(* Logix 5000 project; controller HP_SSC01 vendor 1 type 14 code 67 rev 17.7; software revision 17.01; part 2 of 15 *)
(* tags used below, declared in another part *)
   A_C1_0300 : ALIAS FOR C1_FaultStandard.0;
   A_C1_0301 : ALIAS FOR C1_FaultStandard.1;
   A_C1_0302 : ALIAS FOR C1_FaultStandard.2;
   A_C1_0303 : ALIAS FOR C1_FaultStandard.3;
   A_C1_0305 : ALIAS FOR C1_FaultStandard.5;
   A_C1_0309 : ALIAS FOR C1_FaultStandard.9;
   A_C1_0310 : ALIAS FOR C1_FaultStandard.10;
   A_C1_0311 : ALIAS FOR C1_FaultStandard.11;
   A_C1_0312 : ALIAS FOR C1_FaultStandard.12;
   A_C1_0313 : ALIAS FOR C1_FaultStandard.13;
   A_C1_0314 : ALIAS FOR C1_FaultStandard.14;
   A_C1_0315 : ALIAS FOR C1_FaultStandard.15;
   A_C1_0317 : ALIAS FOR C1_FaultStandard.17;
   A_C1_0319 : ALIAS FOR C1_FaultStandard.19;
   A_C1_0321 : ALIAS FOR C1_FaultStandard.21;
   A_C1_0322 : ALIAS FOR C1_FaultStandard.22;
   A_C1_0323 : ALIAS FOR C1_FaultStandard.23;
   A_C1_0324 : ALIAS FOR C1_FaultStandard.24;
   A_C1_0325 : ALIAS FOR C1_FaultStandard.25;
   A_C1_0327 : ALIAS FOR C1_FaultStandard.27;
   A_C1_0328 : ALIAS FOR C1_FaultStandard.28;
   A_C1_0329 : ALIAS FOR C1_FaultStandard.29;
   A_C1_0330 : ALIAS FOR C1_FaultStandard.30;
   A_C1_0331 : ALIAS FOR C1_FaultStandard.31;
   A_C1_0404 : ALIAS FOR C1_Warning.4;
   A_C1_0406 : ALIAS FOR C1_Warning.6;
   A_C1_0407 : ALIAS FOR C1_Warning.7;
   A_C1_0408 : ALIAS FOR C1_Warning.8;
   A_C1_0409 : ALIAS FOR C1_Warning.9;
   A_C1_0412 : ALIAS FOR C1_Warning.12;
   A_C1_0413 : ALIAS FOR C1_Warning.13;
   A_C1_0414 : ALIAS FOR C1_Warning.14;
   A_C1_0415 : ALIAS FOR C1_Warning.15;
   A_C1_0416 : ALIAS FOR C1_Warning.16;
   A_C1_0424 : ALIAS FOR C1_Warning.24;
   A_C1_0427 : ALIAS FOR C1_Warning.27;
   A_C1_0428 : ALIAS FOR C1_Warning.28;
   A_C1_0430 : ALIAS FOR C1_Warning.30;
   C1 : AXIS_SERVO_DRIVE;
   C1_32HourTimers : TIMER[8];
   C1_All_DLY_OK : BOOL;
   C1_BrakeSequenceInProcess : BOOL;
   C1_BrakeTest : BOOL;
   C1_BrakeTestEndPosition : REAL;
   C1_BrakeTestFailed : BOOL;
   C1_BrakeTestLocalDisable : BOOL;
   C1_BrakeTestMAJ01 : MOTION_INSTRUCTION;
   C1_BrakeTestMessageNumber : DINT;
   C1_BrakeTestONS : BOOL;
   C1_BrakeTestSelected : BOOL;
   C1_BrakeTestSequence : DINT;
   C1_BrakeTestSequenceAlarms : DINT;
   C1_BrakeTestSequenceAlarmTimer : TIMER[16];
   C1_BrakeTestSequenceONS : DINT;
   C1_BrakeTestStartPosition : REAL;
   C1_BrakeTestStoppingDistance : REAL;
   C1_BrakeTestTimerHoldVel : TIMER;
   C1_BrakeTestWarning : BOOL;
   C1_DisableTimer : TIMER;
   C1_DumpTest : BOOL;
   C1_DumpValveFailedOff : BOOL;
   C1_DumpValveFailedOn : BOOL;
   C1_DumpValveMessageNumber : DINT;
   C1_DumpValveTestDelay : TIMER[4];
   C1_DumpValveTestDelay2 : TIMER;
   C1_DumpValveTestSelected : BOOL;
   C1_DumpValveTestSequence : DINT;
   C1_DumpValveTestSequenceAlarms : DINT;
   C1_DumpValveTestSequenceAlarmTimer : TIMER[16];
   C1_EncoderCounts : DINT;
   C1_EncoderCountsRaw : ALIAS FOR C1_RIO_AENT:3:I.PresentData;
   C1_EncoderDegree : REAL;
   C1_FaultDebounce : TIMER[16];
   C1_FaultHoldTimer : TIMER[8];
   C1_FaultHomeSwitchNotFound : BOOL;
   C1_FaultStandard : DINT;
   C1_HomeInputStatus : BOOL;
   C1_HomeSequence : DINT;
   C1_HomeSequenceAlarms : DINT;
   C1_HomeSwitchFaultK7KFailedOff : BOOL;
   C1_HomeSwitchFaultK7KFailedOn : BOOL;
   C1_HomeSwitchFaultSafeFailedOff : BOOL;
   C1_HomeSwitchFaultSafeFailedOn : BOOL;
   C1_IndexEnable : BOOL;
   C1_JogEnable : BOOL;
   C1_LIM_ALARM_B : ALIAS FOR C1_RIO_AENT:I.Data[1].0;
   C1_MaintEnable : BOOL;
   C1_MotorActualPositionX1000 : DINT;
   C1_MotorAverageVelocityX1000 : DINT;
   C1_MotorFan : ALIAS FOR C1_RIO_AENT:O.Data[2].0;
   C1_MSF : MOTION_INSTRUCTION;
   C1_MSO : MOTION_INSTRUCTION;
   C1_OIT_Current : DINT;
   C1_ONS_Fault : DINT;
   C1_RemoteBrakeAndHomeSequenceAlarms : DINT;
   C1_RemoteBrakeTestCMD : BOOL;
   C1_RemoteDumpTestCMD : BOOL;
   C1_ServoActionStatusOffDelay : TIMER;
   C1_ServoActionStatusOnDelay : TIMER;
   C1_ServoFanOverload : ALIAS FOR C1_RIO_AENT:I.Data[1].2;
   C1_SS_LocalRemote_1_IsRemote : ALIAS FOR C1_RIO_AENT:1:I.3;
   C1_SS_RemoteMode : BOOL;
   C1_Warning : DINT;
   C1DumpValveTestSequenceONS : DINT;
   RCS_CMD_RunInAuto : BOOL;
   RCS_SyncMotionEnable : BOOL;
   S_C1_EncoderPositionDegree : DINT;
   S_C1_ExecutePB : BOOL;
   S_C1_FaultReset : BOOL;
   S_C1_ModeLocal : BOOL;
   S_C1_ModeRemote : BOOL;
   S_C1_MotionEnabled : BOOL;
   S_C1_MSTOP_InputOK : BOOL;
   S_C1_NearOnPath : BOOL;
   S_C1_OffPath : BOOL;
   S_C1_OIT_FaultReset : BOOL;
   S_C1_OutputEnable : BOOL;
   S_C1_PressureOK : ALIAS FOR C1_Safe:I.Pt05Data;
   S_C1_SAFETY_ENABLE_1 : ALIAS FOR C1_Safe:O.Pt00Data;
   S_C1_SAFETY_ENABLE_2 : ALIAS FOR C1_Safe:O.Pt01Data;
   S_C1_Stop1_OK : BOOL;
   S_RCS_CMD_FaultReset : BOOL;
   STS_Enable_Rail : DINT;
   ZZZ_DIAG_A_C1_0302 : BOOL;
   ZZZ_DIAG_C1_AxisFault : DINT;
   ZZZ_DIAG_C1_AxisStatus : DINT;
   ZZZ_DIAG_C1_EnableRail : DINT;
   ZZZ_DIAG_C1_MotionStatus : DINT;
   ZZZ_DIAG_C1_MSF : MOTION_INSTRUCTION;
   ZZZ_DIAG_C1_MSO : MOTION_INSTRUCTION;
   ZZZ_DIAG_C1_OneTimeOnly : BOOL;
   ZZZ_DIAG_C1_OutputEnable : BOOL;
   ZZZ_DIAG_C1_OutputEnable_ACC : DINT;
   ZZZ_DIAG_ONS : DINT;
   ZZZ_DIAG_S_C1_OutputEnableTON : TIMER;
   ZZZ_DIAG_S_C1_SAFETY_ENABLE_1 : BOOL;
   ZZZ_DIAG_S_C1_SAFETY_ENABLE_2 : BOOL;

PROGRAM Carousel1   (* main routine C100_Main *)
VAR
   SCRV_01 : S_CURVE := (In := 26.237068, AccelRate := 100000.0, DecelRate := 100000.0, JerkRate := 100.0, RTSTime := 1, S_Mode := 1, Out := 25.846554, Rate := 8.784333, DeltaT := 0.01);
   zzz_Test10 : BOOL;
   zzz_Test11 : BOOL;
   zzz_TestOffset : DINT := 1000;
   zzz_TestWord10 : DINT;
END_VAR

ROUTINE C100_Main   (* ladder *)
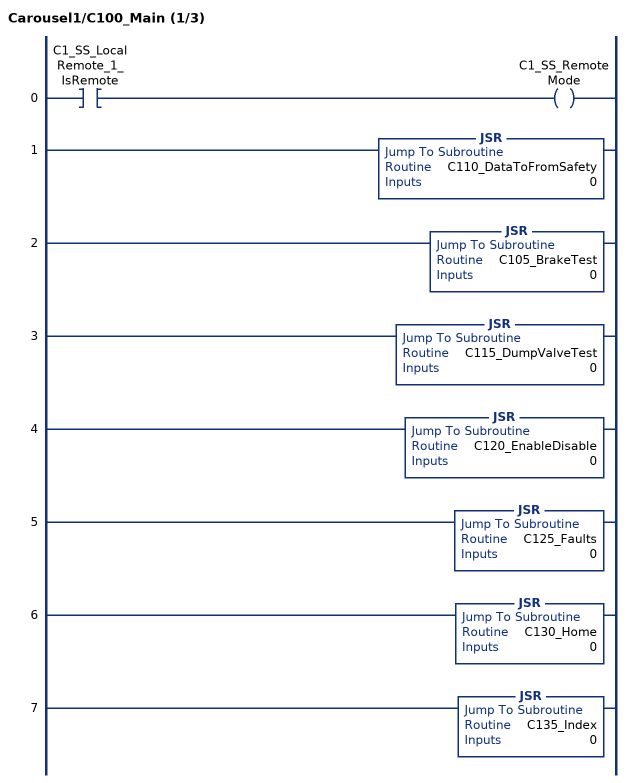
   0: XIC(C1_SS_LocalRemote_1_IsRemote)OTE(C1_SS_RemoteMode);
   1: JSR(C110_DataToFromSafety,0);
   2: JSR(C105_BrakeTest,0);
   3: JSR(C115_DumpValveTest,0);
   4: JSR(C120_EnableDisable,0);
   5: JSR(C125_Faults,0);
   6: JSR(C130_Home,0);
   7: JSR(C135_Index,0);
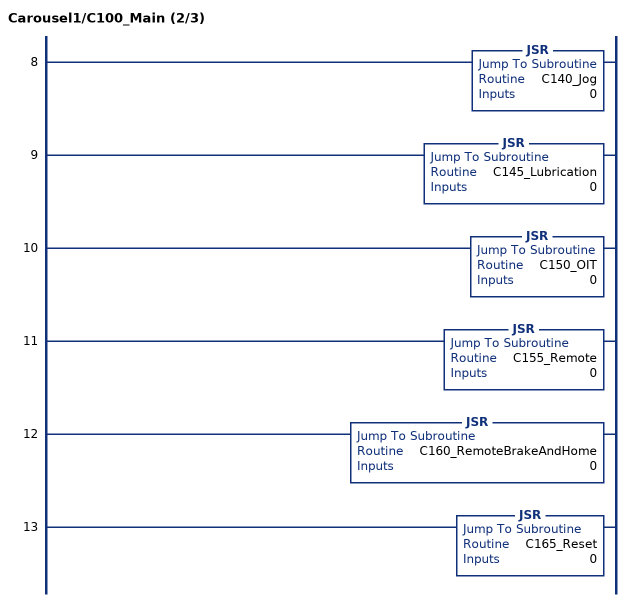
   8: JSR(C140_Jog,0);
   9: JSR(C145_Lubrication,0);
   10: JSR(C150_OIT,0);
   11: JSR(C155_Remote,0);
   12: JSR(C160_RemoteBrakeAndHome,0);
   13: JSR(C165_Reset,0);
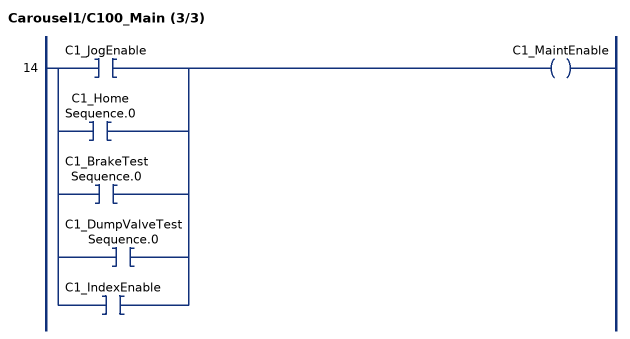
   14: [XIC(C1_JogEnable) ,XIC(C1_HomeSequence.0) ,XIC(C1_BrakeTestSequence.0) ,XIC(C1_DumpValveTestSequence.0) ,XIC(C1_IndexEnable) ]OTE(C1_MaintEnable);
END_ROUTINE

ROUTINE C105_BrakeTest   (* ladder *)
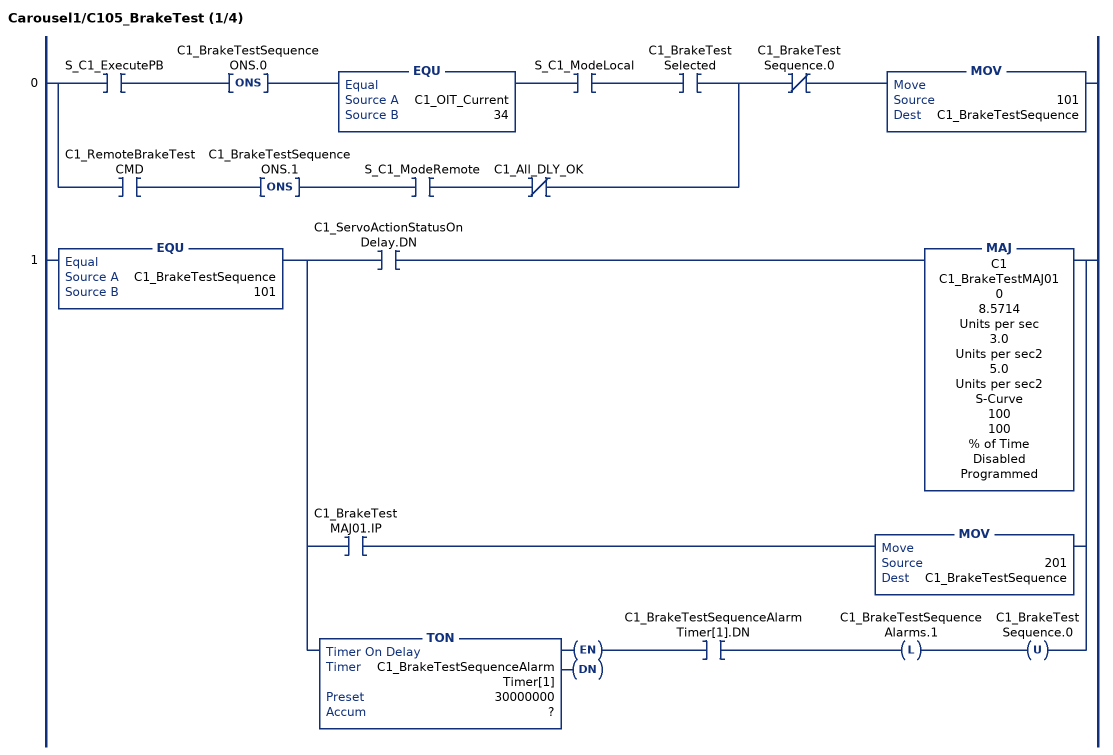
   0: [XIC(S_C1_ExecutePB) ONS(C1_BrakeTestSequenceONS.0) EQU(C1_OIT_Current,34) XIC(S_C1_ModeLocal) XIC(C1_BrakeTestSelected) ,XIC(C1_RemoteBrakeTestCMD) ONS(C1_BrakeTestSequenceONS.1) XIC(S_C1_ModeRemote) XIO(C1_All_DLY_OK) ]XIO(C1_BrakeTestSequence.0)MOV(101,C1_BrakeTestSequence);
   1: EQU(C1_BrakeTestSequence,101)[XIC(C1_ServoActionStatusOnDelay.DN) MAJ(C1,C1_BrakeTestMAJ01,0,8.5714,Units per sec,3.0,Units per sec2,5.0,Units per sec2,S-Curve,100,100,% of Time,Disabled,Programmed) ,XIC(C1_BrakeTestMAJ01.IP) MOV(201,C1_BrakeTestSequence) ,TON(C1_BrakeTestSequenceAlarmTimer[1],?,?) XIC(C1_BrakeTestSequenceAlarmTimer[1].DN) OTL(C1_BrakeTestSequenceAlarms.1) OTU(C1_BrakeTestSequence.0) ];
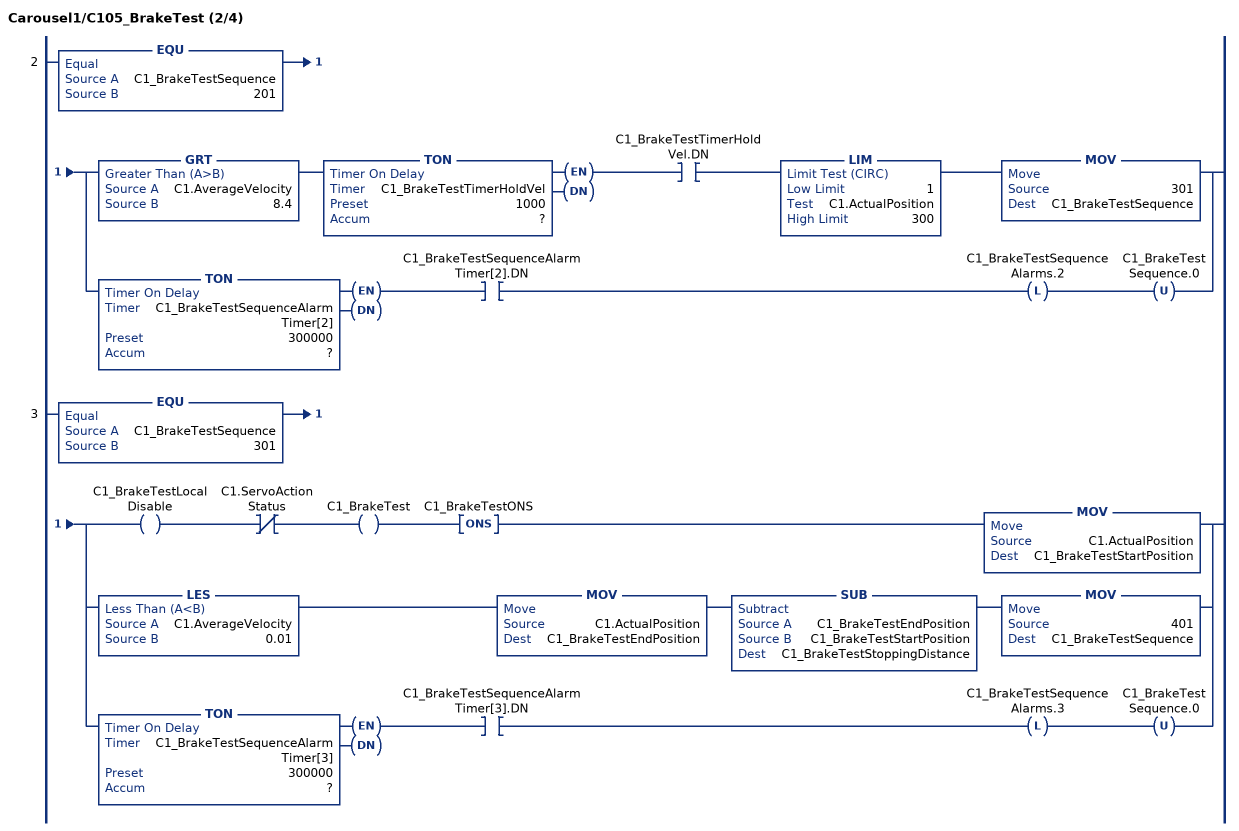
   2: EQU(C1_BrakeTestSequence,201)[GRT(C1.AverageVelocity,8.4) TON(C1_BrakeTestTimerHoldVel,?,?) XIC(C1_BrakeTestTimerHoldVel.DN) LIM(1,C1.ActualPosition,300) MOV(301,C1_BrakeTestSequence) ,TON(C1_BrakeTestSequenceAlarmTimer[2],?,?) XIC(C1_BrakeTestSequenceAlarmTimer[2].DN) OTL(C1_BrakeTestSequenceAlarms.2) OTU(C1_BrakeTestSequence.0) ];
   3: EQU(C1_BrakeTestSequence,301)[OTE(C1_BrakeTestLocalDisable) XIO(C1.ServoActionStatus) OTE(C1_BrakeTest) ONS(C1_BrakeTestONS) MOV(C1.ActualPosition,C1_BrakeTestStartPosition) ,LES(C1.AverageVelocity,0.01) MOV(C1.ActualPosition,C1_BrakeTestEndPosition) SUB(C1_BrakeTestEndPosition,C1_BrakeTestStartPosition,C1_BrakeTestStoppingDistance) MOV(401,C1_BrakeTestSequence) ,TON(C1_BrakeTestSequenceAlarmTimer[3],?,?) XIC(C1_BrakeTestSequenceAlarmTimer[3].DN) OTL(C1_BrakeTestSequenceAlarms.3) OTU(C1_BrakeTestSequence.0) ];
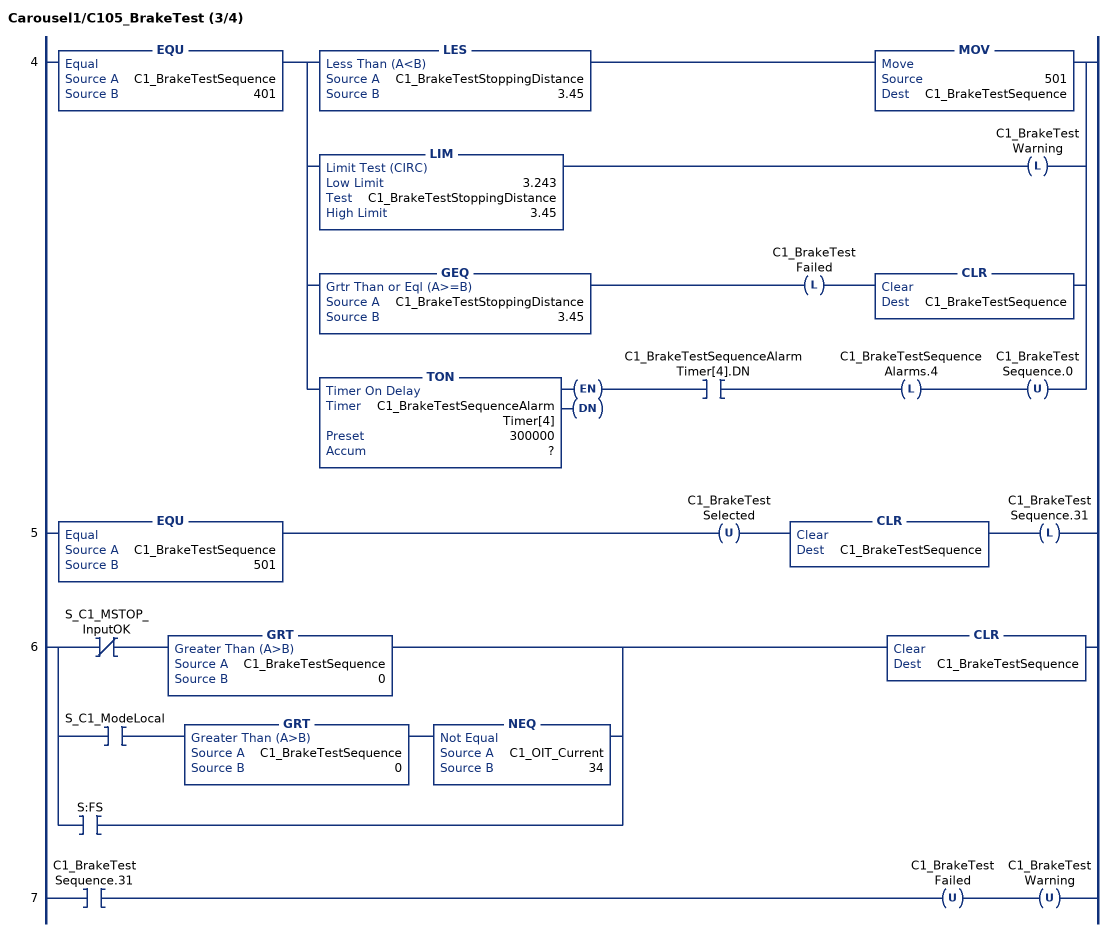
   4: EQU(C1_BrakeTestSequence,401)[LES(C1_BrakeTestStoppingDistance,3.45) MOV(501,C1_BrakeTestSequence) ,LIM(3.243,C1_BrakeTestStoppingDistance,3.45) OTL(C1_BrakeTestWarning) ,GEQ(C1_BrakeTestStoppingDistance,3.45) OTL(C1_BrakeTestFailed) CLR(C1_BrakeTestSequence) ,TON(C1_BrakeTestSequenceAlarmTimer[4],?,?) XIC(C1_BrakeTestSequenceAlarmTimer[4].DN) OTL(C1_BrakeTestSequenceAlarms.4) OTU(C1_BrakeTestSequence.0) ];
   5: EQU(C1_BrakeTestSequence,501)OTU(C1_BrakeTestSelected)CLR(C1_BrakeTestSequence)OTL(C1_BrakeTestSequence.31);
   6: [XIO(S_C1_MSTOP_InputOK) GRT(C1_BrakeTestSequence,0) ,XIC(S_C1_ModeLocal) GRT(C1_BrakeTestSequence,0) NEQ(C1_OIT_Current,34) ,XIC(S:FS) ]CLR(C1_BrakeTestSequence);
   7: XIC(C1_BrakeTestSequence.31)OTU(C1_BrakeTestFailed)OTU(C1_BrakeTestWarning);
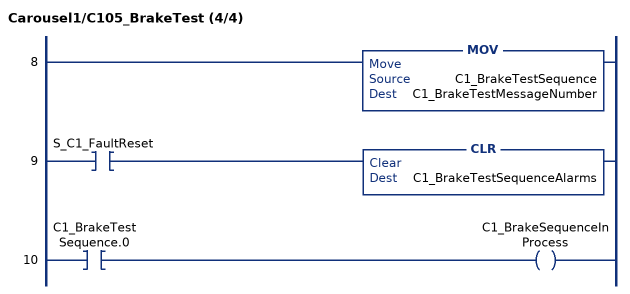
   8: MOV(C1_BrakeTestSequence,C1_BrakeTestMessageNumber);
   9: XIC(S_C1_FaultReset)CLR(C1_BrakeTestSequenceAlarms);
   10: XIC(C1_BrakeTestSequence.0)OTE(C1_BrakeSequenceInProcess);
END_ROUTINE

ROUTINE C110_DataToFromSafety   (* ladder *)
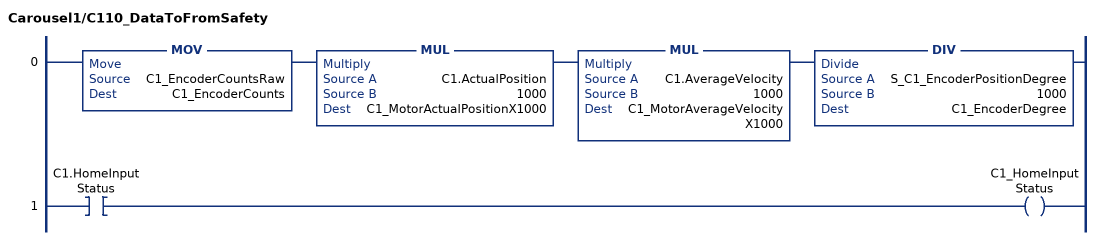
   0: MOV(C1_EncoderCountsRaw,C1_EncoderCounts)MUL(C1.ActualPosition,1000,C1_MotorActualPositionX1000)MUL(C1.AverageVelocity,1000,C1_MotorAverageVelocityX1000)DIV(S_C1_EncoderPositionDegree,1000,C1_EncoderDegree);
   1: XIC(C1.HomeInputStatus)OTE(C1_HomeInputStatus);
END_ROUTINE

ROUTINE C115_DumpValveTest   (* ladder *)
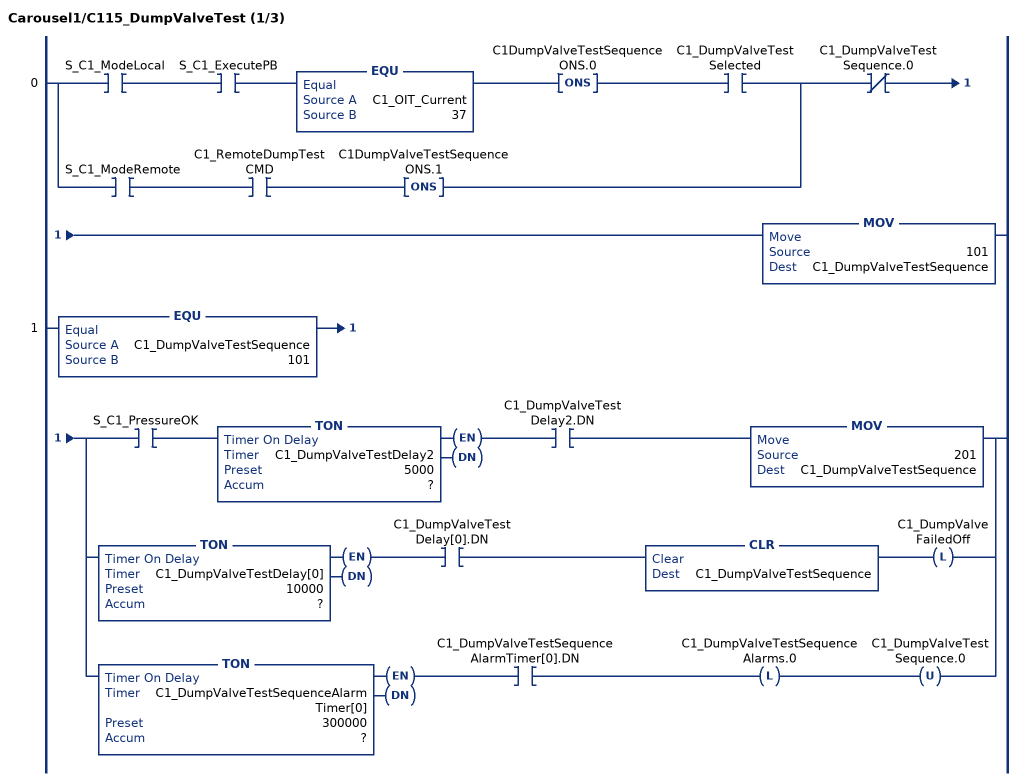
   0: [XIC(S_C1_ModeLocal) XIC(S_C1_ExecutePB) EQU(C1_OIT_Current,37) ONS(C1DumpValveTestSequenceONS.0) XIC(C1_DumpValveTestSelected) ,XIC(S_C1_ModeRemote) XIC(C1_RemoteDumpTestCMD) ONS(C1DumpValveTestSequenceONS.1) ]XIO(C1_DumpValveTestSequence.0)MOV(101,C1_DumpValveTestSequence);
   1: EQU(C1_DumpValveTestSequence,101)[XIC(S_C1_PressureOK) TON(C1_DumpValveTestDelay2,?,?) XIC(C1_DumpValveTestDelay2.DN) MOV(201,C1_DumpValveTestSequence) ,TON(C1_DumpValveTestDelay[0],?,?) XIC(C1_DumpValveTestDelay[0].DN) CLR(C1_DumpValveTestSequence) OTL(C1_DumpValveFailedOff) ,TON(C1_DumpValveTestSequenceAlarmTimer[0],?,?) XIC(C1_DumpValveTestSequenceAlarmTimer[0].DN) OTL(C1_DumpValveTestSequenceAlarms.0) OTU(C1_DumpValveTestSequence.0) ];
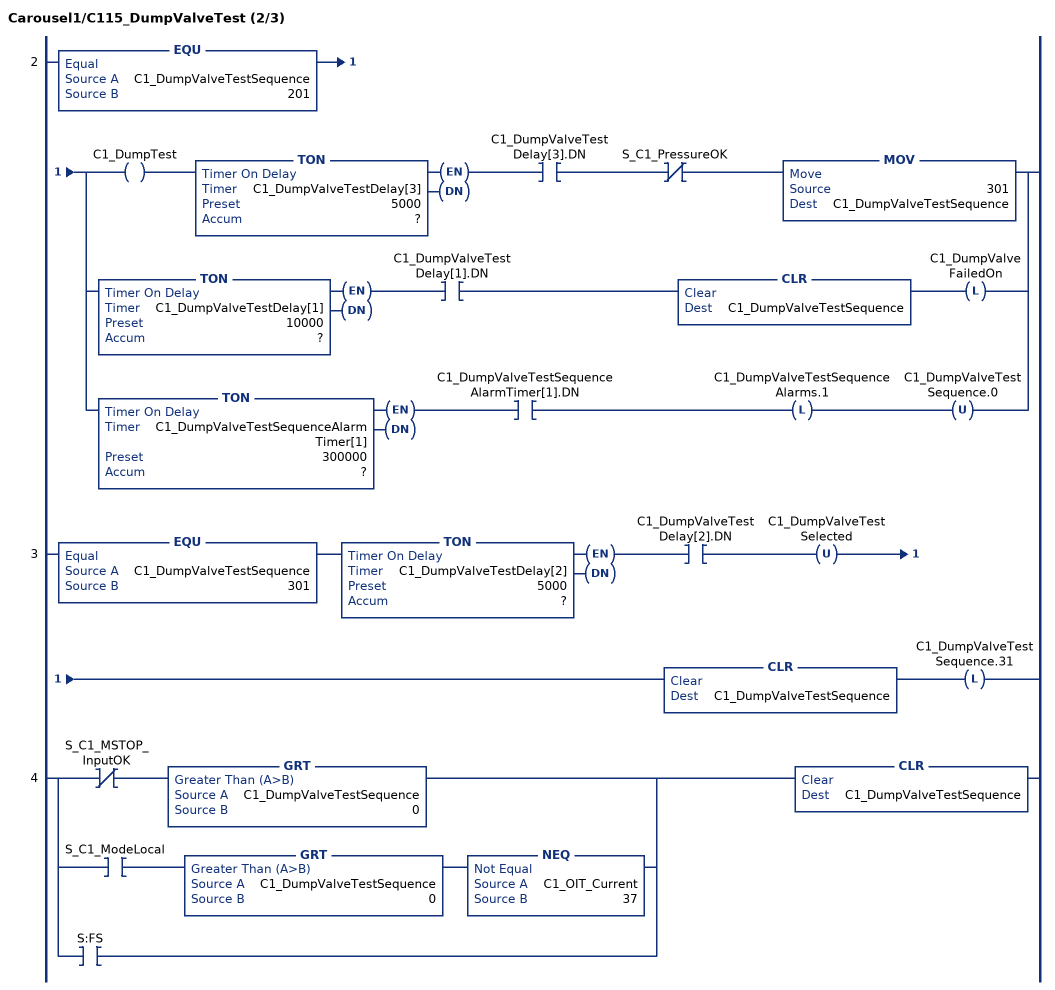
   2: EQU(C1_DumpValveTestSequence,201)[OTE(C1_DumpTest) TON(C1_DumpValveTestDelay[3],?,?) XIC(C1_DumpValveTestDelay[3].DN) XIO(S_C1_PressureOK) MOV(301,C1_DumpValveTestSequence) ,TON(C1_DumpValveTestDelay[1],?,?) XIC(C1_DumpValveTestDelay[1].DN) CLR(C1_DumpValveTestSequence) OTL(C1_DumpValveFailedOn) ,TON(C1_DumpValveTestSequenceAlarmTimer[1],?,?) XIC(C1_DumpValveTestSequenceAlarmTimer[1].DN) OTL(C1_DumpValveTestSequenceAlarms.1) OTU(C1_DumpValveTestSequence.0) ];
   3: EQU(C1_DumpValveTestSequence,301)TON(C1_DumpValveTestDelay[2],?,?)XIC(C1_DumpValveTestDelay[2].DN)OTU(C1_DumpValveTestSelected)CLR(C1_DumpValveTestSequence)OTL(C1_DumpValveTestSequence.31);
   4: [XIO(S_C1_MSTOP_InputOK) GRT(C1_DumpValveTestSequence,0) ,XIC(S_C1_ModeLocal) GRT(C1_DumpValveTestSequence,0) NEQ(C1_OIT_Current,37) ,XIC(S:FS) ]CLR(C1_DumpValveTestSequence);
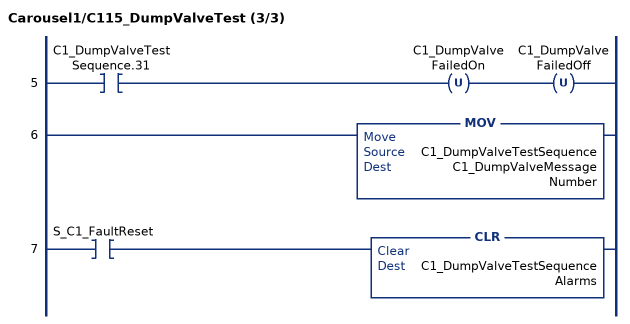
   5: XIC(C1_DumpValveTestSequence.31)OTU(C1_DumpValveFailedOn)OTU(C1_DumpValveFailedOff);
   6: MOV(C1_DumpValveTestSequence,C1_DumpValveMessageNumber);
   7: XIC(S_C1_FaultReset)CLR(C1_DumpValveTestSequenceAlarms);
END_ROUTINE

ROUTINE C120_EnableDisable   (* ladder *)
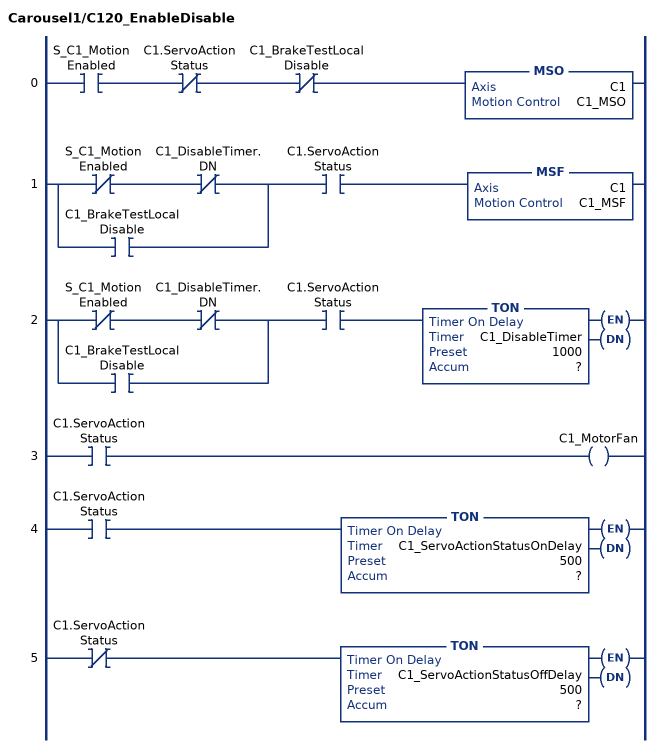
   0: XIC(S_C1_MotionEnabled)XIO(C1.ServoActionStatus)XIO(C1_BrakeTestLocalDisable)MSO(C1,C1_MSO);
   1: [XIO(S_C1_MotionEnabled) XIO(C1_DisableTimer.DN) ,XIC(C1_BrakeTestLocalDisable) ]XIC(C1.ServoActionStatus)MSF(C1,C1_MSF);
   2: [XIO(S_C1_MotionEnabled) XIO(C1_DisableTimer.DN) ,XIC(C1_BrakeTestLocalDisable) ]XIC(C1.ServoActionStatus)TON(C1_DisableTimer,?,?);
   3: XIC(C1.ServoActionStatus)OTE(C1_MotorFan);
   4: XIC(C1.ServoActionStatus)TON(C1_ServoActionStatusOnDelay,?,?);
   5: XIO(C1.ServoActionStatus)TON(C1_ServoActionStatusOffDelay,?,?);
END_ROUTINE

ROUTINE C125_Faults   (* ladder *)
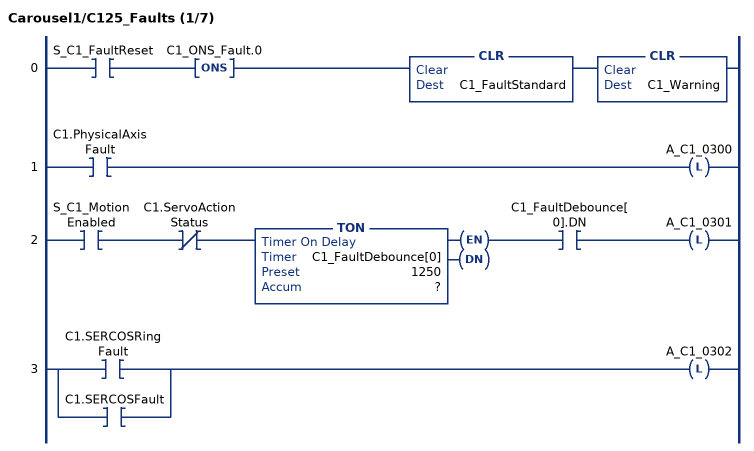
   0: XIC(S_C1_FaultReset)ONS(C1_ONS_Fault.0)CLR(C1_FaultStandard)CLR(C1_Warning);
   1: XIC(C1.PhysicalAxisFault)OTL(A_C1_0300);
   2: XIC(S_C1_MotionEnabled)XIO(C1.ServoActionStatus)TON(C1_FaultDebounce[0],?,?)XIC(C1_FaultDebounce[0].DN)OTL(A_C1_0301);
   3: [XIC(C1.SERCOSRingFault) ,XIC(C1.SERCOSFault) ]OTL(A_C1_0302);
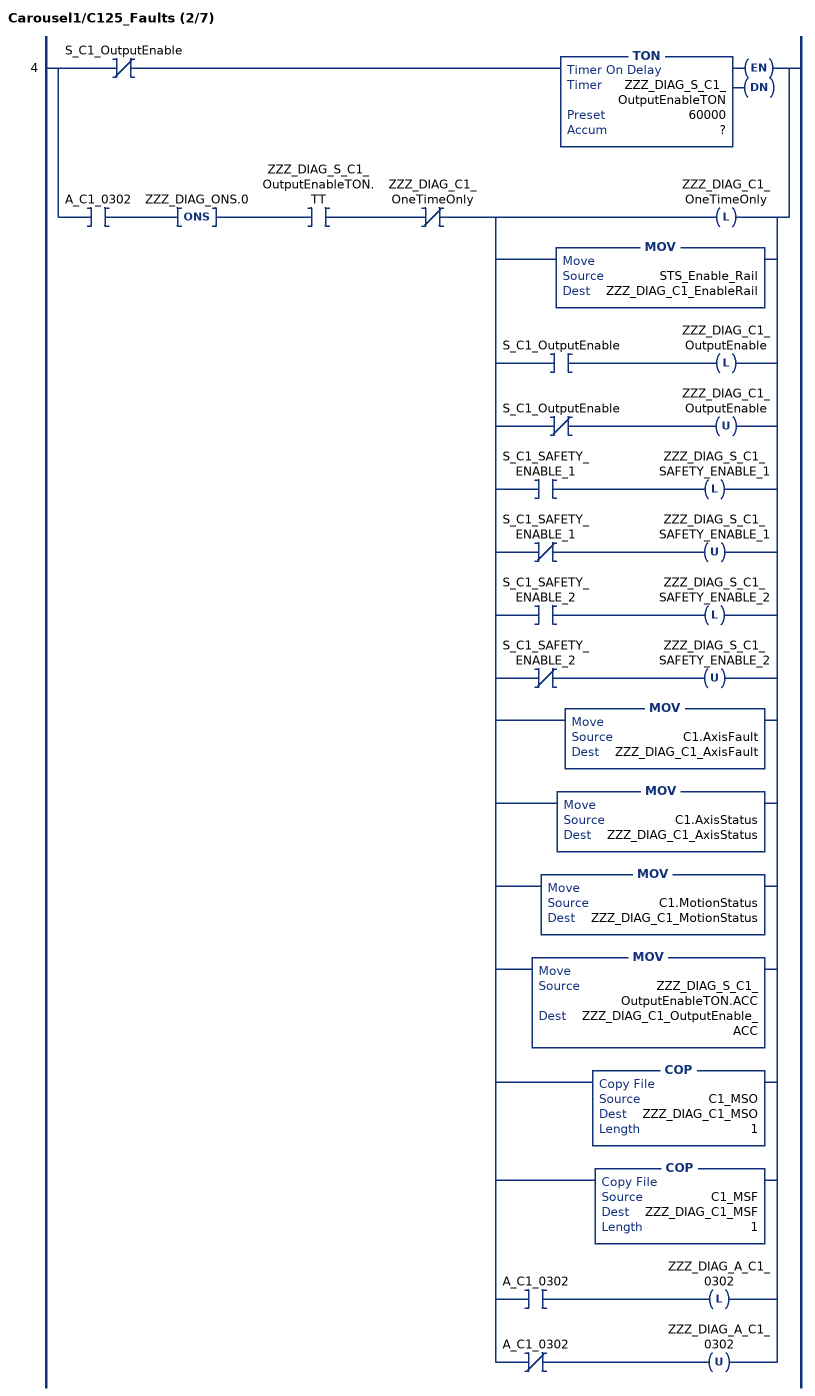
   4: [XIO(S_C1_OutputEnable) TON(ZZZ_DIAG_S_C1_OutputEnableTON,?,?) ,XIC(A_C1_0302) ONS(ZZZ_DIAG_ONS.0) XIC(ZZZ_DIAG_S_C1_OutputEnableTON.TT) XIO(ZZZ_DIAG_C1_OneTimeOnly) [OTL(ZZZ_DIAG_C1_OneTimeOnly) ,MOV(STS_Enable_Rail,ZZZ_DIAG_C1_EnableRail) ,XIC(S_C1_OutputEnable) OTL(ZZZ_DIAG_C1_OutputEnable) ,XIO(S_C1_OutputEnable) OTU(ZZZ_DIAG_C1_OutputEnable) ,XIC(S_C1_SAFETY_ENABLE_1) OTL(ZZZ_DIAG_S_C1_SAFETY_ENABLE_1) ,XIO(S_C1_SAFETY_ENABLE_1) OTU(ZZZ_DIAG_S_C1_SAFETY_ENABLE_1) ,XIC(S_C1_SAFETY_ENABLE_2) OTL(ZZZ_DIAG_S_C1_SAFETY_ENABLE_2) ,XIO(S_C1_SAFETY_ENABLE_2) OTU(ZZZ_DIAG_S_C1_SAFETY_ENABLE_2) ,MOV(C1.AxisFault,ZZZ_DIAG_C1_AxisFault) ,MOV(C1.AxisStatus,ZZZ_DIAG_C1_AxisStatus) ,MOV(C1.MotionStatus,ZZZ_DIAG_C1_MotionStatus) ,MOV(ZZZ_DIAG_S_C1_OutputEnableTON.ACC,ZZZ_DIAG_C1_OutputEnable_ACC) ,COP(C1_MSO,ZZZ_DIAG_C1_MSO,1) ,COP(C1_MSF,ZZZ_DIAG_C1_MSF,1) ,XIC(A_C1_0302) OTL(ZZZ_DIAG_A_C1_0302) ,XIO(A_C1_0302) OTU(ZZZ_DIAG_A_C1_0302) ] ];
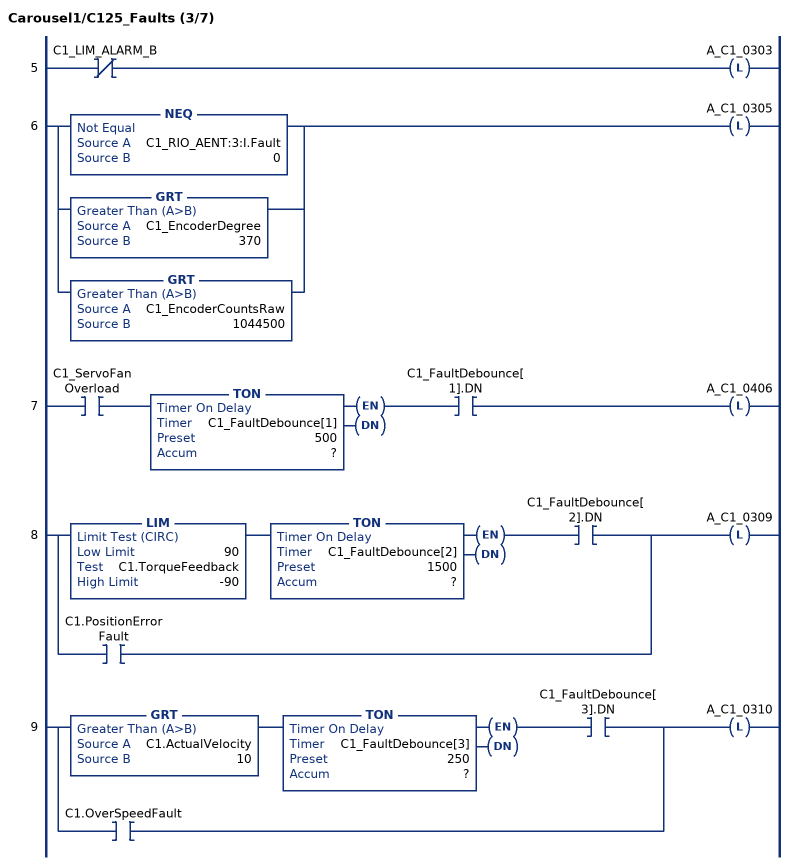
   5: XIO(C1_LIM_ALARM_B)OTL(A_C1_0303);
   6: [NEQ(C1_RIO_AENT:3:I.Fault,0) ,GRT(C1_EncoderDegree,370) ,GRT(C1_EncoderCountsRaw,1044500) ]OTL(A_C1_0305);
   7: XIC(C1_ServoFanOverload)TON(C1_FaultDebounce[1],?,?)XIC(C1_FaultDebounce[1].DN)OTL(A_C1_0406);
   8: [LIM(90,C1.TorqueFeedback,-90) TON(C1_FaultDebounce[2],?,?) XIC(C1_FaultDebounce[2].DN) ,XIC(C1.PositionErrorFault) ]OTL(A_C1_0309);
   9: [GRT(C1.ActualVelocity,10) TON(C1_FaultDebounce[3],?,?) XIC(C1_FaultDebounce[3].DN) ,XIC(C1.OverSpeedFault) ]OTL(A_C1_0310);
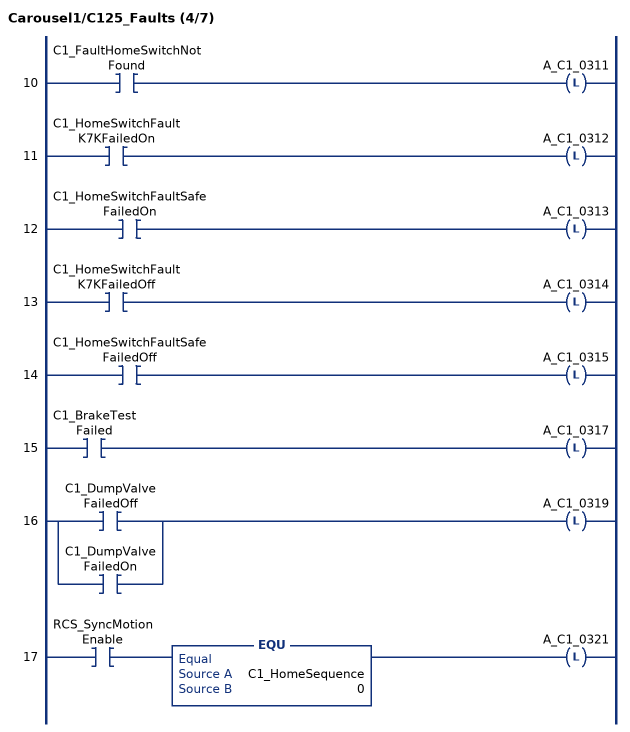
   10: XIC(C1_FaultHomeSwitchNotFound)OTL(A_C1_0311);
   11: XIC(C1_HomeSwitchFaultK7KFailedOn)OTL(A_C1_0312);
   12: XIC(C1_HomeSwitchFaultSafeFailedOn)OTL(A_C1_0313);
   13: XIC(C1_HomeSwitchFaultK7KFailedOff)OTL(A_C1_0314);
   14: XIC(C1_HomeSwitchFaultSafeFailedOff)OTL(A_C1_0315);
   15: XIC(C1_BrakeTestFailed)OTL(A_C1_0317);
   16: [XIC(C1_DumpValveFailedOff) ,XIC(C1_DumpValveFailedOn) ]OTL(A_C1_0319);
   17: XIC(RCS_SyncMotionEnable)EQU(C1_HomeSequence,0)OTL(A_C1_0321);
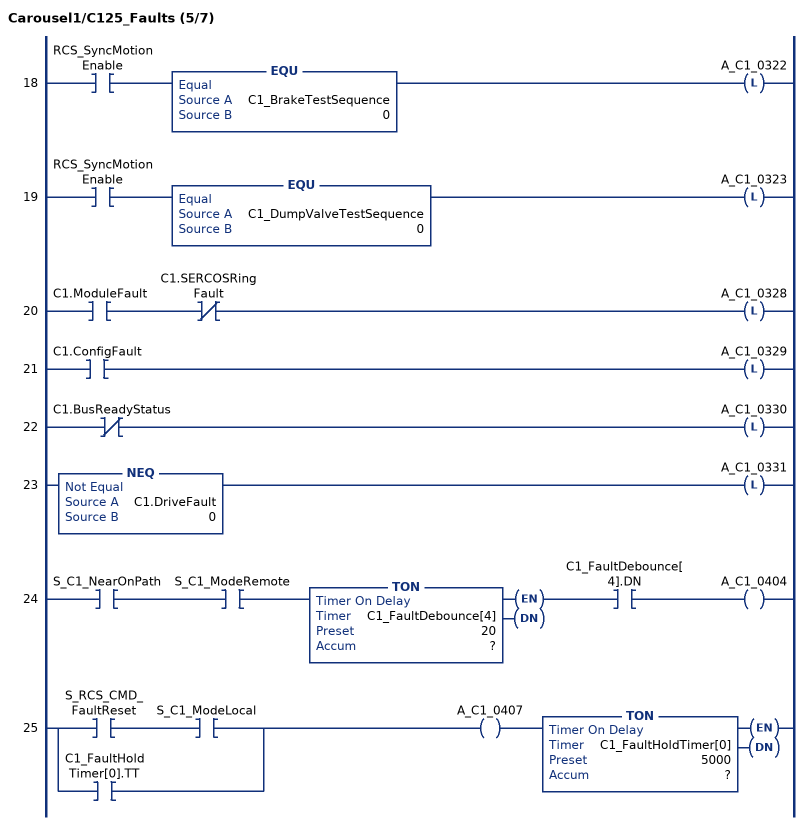
   18: XIC(RCS_SyncMotionEnable)EQU(C1_BrakeTestSequence,0)OTL(A_C1_0322);
   19: XIC(RCS_SyncMotionEnable)EQU(C1_DumpValveTestSequence,0)OTL(A_C1_0323);
   20: XIC(C1.ModuleFault)XIO(C1.SERCOSRingFault)OTL(A_C1_0328);
   21: XIC(C1.ConfigFault)OTL(A_C1_0329);
   22: XIO(C1.BusReadyStatus)OTL(A_C1_0330);
   23: NEQ(C1.DriveFault,0)OTL(A_C1_0331);
   24: XIC(S_C1_NearOnPath)XIC(S_C1_ModeRemote)TON(C1_FaultDebounce[4],?,?)XIC(C1_FaultDebounce[4].DN)OTE(A_C1_0404);
   25: [XIC(S_RCS_CMD_FaultReset) XIC(S_C1_ModeLocal) ,XIC(C1_FaultHoldTimer[0].TT) ]OTE(A_C1_0407)TON(C1_FaultHoldTimer[0],?,?);
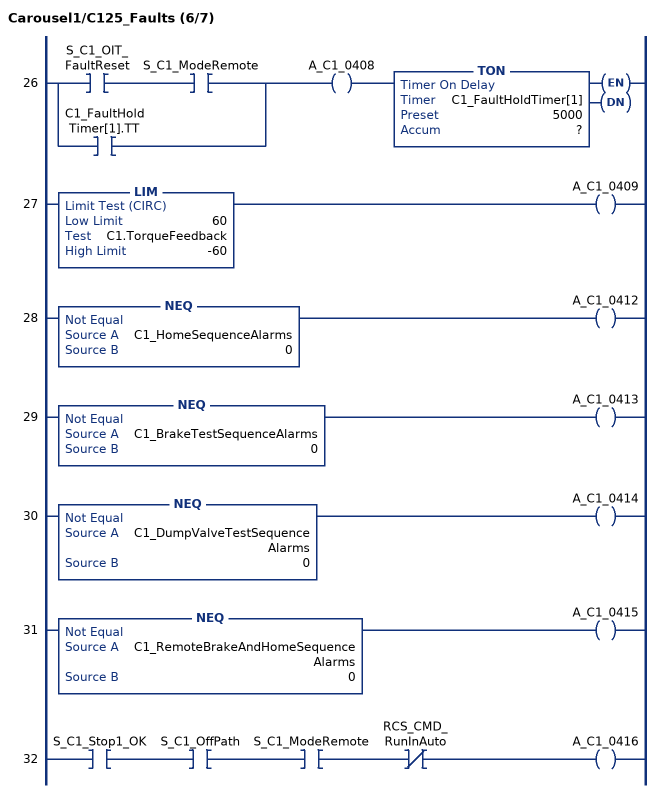
   26: [XIC(S_C1_OIT_FaultReset) XIC(S_C1_ModeRemote) ,XIC(C1_FaultHoldTimer[1].TT) ]OTE(A_C1_0408)TON(C1_FaultHoldTimer[1],?,?);
   27: LIM(60,C1.TorqueFeedback,-60)OTE(A_C1_0409);
   28: NEQ(C1_HomeSequenceAlarms,0)OTE(A_C1_0412);
   29: NEQ(C1_BrakeTestSequenceAlarms,0)OTE(A_C1_0413);
   30: NEQ(C1_DumpValveTestSequenceAlarms,0)OTE(A_C1_0414);
   31: NEQ(C1_RemoteBrakeAndHomeSequenceAlarms,0)OTE(A_C1_0415);
   32: XIC(S_C1_Stop1_OK)XIC(S_C1_OffPath)XIC(S_C1_ModeRemote)XIO(RCS_CMD_RunInAuto)OTE(A_C1_0416);
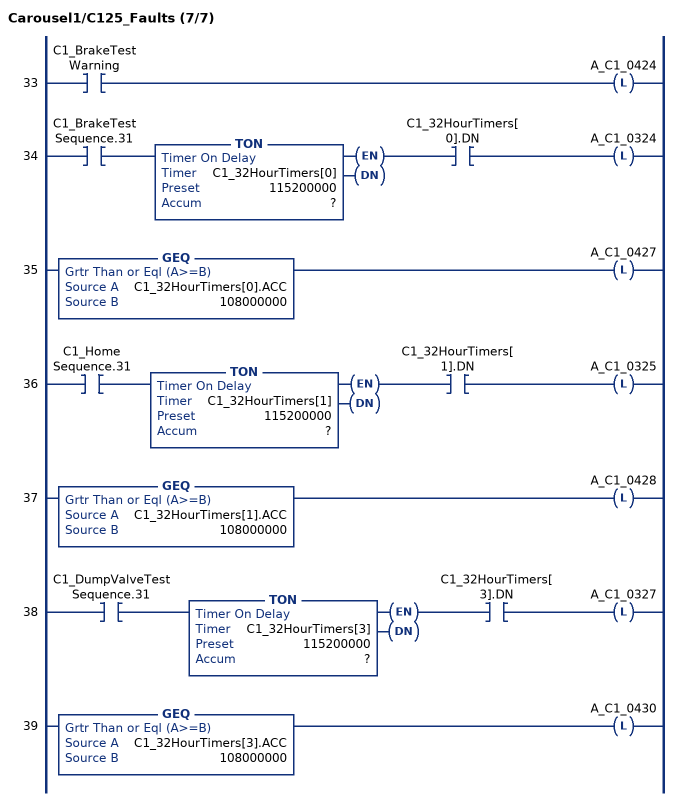
   33: XIC(C1_BrakeTestWarning)OTL(A_C1_0424);
   34: XIC(C1_BrakeTestSequence.31)TON(C1_32HourTimers[0],?,?)XIC(C1_32HourTimers[0].DN)OTL(A_C1_0324);
   35: GEQ(C1_32HourTimers[0].ACC,108000000)OTL(A_C1_0427);
   36: XIC(C1_HomeSequence.31)TON(C1_32HourTimers[1],?,?)XIC(C1_32HourTimers[1].DN)OTL(A_C1_0325);
   37: GEQ(C1_32HourTimers[1].ACC,108000000)OTL(A_C1_0428);
   38: XIC(C1_DumpValveTestSequence.31)TON(C1_32HourTimers[3],?,?)XIC(C1_32HourTimers[3].DN)OTL(A_C1_0327);
   39: GEQ(C1_32HourTimers[3].ACC,108000000)OTL(A_C1_0430);
END_ROUTINE
